(* Logix 5000 project; controller OptixProdData_Demo vendor 1 type 14 code 164 rev 37.11; software revision 37.00 *)

TASK MainTask (continuous, watchdog 500 ms) : MainProgram

MODULES
   Local : vendor 1 type 14 code 164 (ICP 0, rev 37.11)
END_MODULES

TYPE str_01 :
STRUCT
   LEN : DINT;
   DATA : SINT[1];
END_STRUCT
END_TYPE

TYPE str_50 :   // String with 50 Characters for SQL Stored Procedures
STRUCT
   LEN : DINT;
   DATA : SINT[50];
END_STRUCT
END_TYPE

TYPE str_Date :
STRUCT
   LEN : DINT;
   DATA : SINT[12];
END_STRUCT
END_TYPE

TYPE str_DateTime :
STRUCT
   LEN : DINT;
   DATA : SINT[22];
END_STRUCT
END_TYPE

TYPE str_Time :
STRUCT
   LEN : DINT;
   DATA : SINT[10];
END_STRUCT
END_TYPE

TYPE udt_CycleTimes :
STRUCT
   ProdLine : str_50;   // Production Line Name
   StationID : str_50;   // Station Name
   TS_PLC : str_DateTime;   // PLC Time Stamp in DateTime format "01/01/2025 15:01:01"
   CycleTime : REAL;   // Cycle time in decimal seconds
   CycleTimeAvg : REAL;   // Cycle Time Average for last hour in deimal seconds
   CycleCount : DINT;   // non-reset Cycle Count
END_STRUCT
END_TYPE

TYPE udt_DateTime :   // WallClock structure
STRUCT
   Year : DINT;   // 2xxx
   Month : DINT;   // 1 - 12
   Day : DINT;   // 01 - 31
   Hour : DINT;   // 0 - 23
   Minute : DINT;   // 0 - 59
   Seconds : DINT;   // 0 - 59
   ms : DINT;   // 0 - 999,999
END_STRUCT
END_TYPE

TYPE udt_LineSummary :   // Summary production data to mimic existing white board
STRUCT
   ProdLine : str_50;   // Production Line Name
   Hour : str_Time;   // 24-hour clock time format HH:MM:SS
   Date : str_Date;   // Date in format 01/01/2025
   TargetQty : DINT;   // Target Qty for hour
   ActQty : DINT;   // Actual qty for hour
   TargetAccQty : DINT;   // Target Accumulated Qty
   ActAccQty : DINT;   // Actual Accumulated Qty
END_STRUCT
END_TYPE

TYPE udt_ProdData :   // Summary production data to mimic existing white board
STRUCT
   PLC_TS : str_DateTime;   // Controller Date Time "HH:MM:SS 01/25/2025"
   ProdLine : str_50;   // Production Line Name
   EquipID : str_50;   // Equipment Name
   ProdCount : DINT;   // Production Counter
   CycleAvg : REAL;   // Average Cycle time (seconds per part)
END_STRUCT
END_TYPE

TYPE udt_SPInterface :
STRUCT
   Trans_DN : BOOL;   // Transaction Complete Bit from Optix to PLC
   SQLErrorNum : DINT;   // SQL Error Number if transaction failed
   Trigger : DINT;   // DINT Value to increment to trigger stored procedure in Optix
END_STRUCT
END_TYPE

ADD_ON_INSTRUCTION ParseTime_SQL   (* revision 1.0 *)
VAR_IN_OUT
   TimeStamp : udt_DateTime; {required}
   Date : str_Date; {required}
   Time : str_Time; {required}
   DateTime : str_DateTime; {required}
END_VAR
VAR
   strTemp2 : str_DateTime; {access None}
   strTemp1 : str_DateTime; {access None}
   strTemp : str_DateTime; {access None}
   strYear : str_Date; {access None}
   strDateTime : str_DateTime; {access None}
   strDate : str_Date; {access None}
   strTime : str_Time; {access None}
END_VAR

ROUTINE Logic   (* structured text *)
   DTOS(TimeStamp.Year, strYear);
   //Create Time format
   #region
   //Hour
   IF TimeStamp.Hour<10 then
   	strTemp1:='0';
   	DTOS(TimeStamp.Hour, strTemp2);
   	CONCAT(strTemp1, strTemp2, strTemp);
   	//0h
   else
   	DTOS(TimeStamp.Hour,strTemp);
   	//hh
   end_if;
   
   strTemp1:=':';
   CONCAT(strTemp, strTemp1, strTime);
   //hh:
   
   //Minutes
   IF TimeStamp.Minute<10 then
   	strTemp1:='0';
   	DTOS(TimeStamp.Minute, strTemp2);
   	CONCAT(strTemp1, strTemp2, strTemp);
   	//0m
   else
   	DTOS(TimeStamp.Minute,strTemp);
   	//mm
   end_if;
   
   strTemp1:=':';
   CONCAT(strTime, strTemp, strTime);
   CONCAT(strTime, strTemp1, strTime);
   //hh:mm:
   //Seconds
   IF TimeStamp.Seconds<10 then
   	strTemp1:='0';
   	DTOS(TimeStamp.Seconds, strTemp2);
   	CONCAT(strTemp1, strTemp2, strTemp);
   	//0n
   else
   	DTOS(TimeStamp.Seconds,strTemp);
   	//nn
   end_if;
   #endregion
   //Time
   CONCAT(strTime, strTemp,strTime);
   //hh:mm:ss
   
   //Build Date
   #region
   //Month
   IF TimeStamp.Month<10 then
   	strTemp1:='0';
   	DTOS(TimeStamp.Month, strTemp2);
   	CONCAT(strTemp1, strTemp2, strTemp);
   	//0n
   else
   	DTOS(TimeStamp.Month,strTemp);
   	//mm
   end_if;
   
   strTemp1:='/';
   CONCAT(strTemp, strTemp1, strDate);
   //mm/
   
   //Day
   IF TimeStamp.Day<10 then
   	strTemp1:='0';
   	DTOS(TimeStamp.Day, strTemp2);
   	CONCAT(strTemp1, strTemp2, strTemp);
   	//0d
   else
   	DTOS(TimeStamp.Day,strTemp);
   	//dd
   end_if;
   strTemp1:='/';
   CONCAT(strDate, strTemp, strDate);
   CONCAT(strDate, strTemp1, strDate);
   //mm/dd/
   #endregion
   //Year
   CONCAT(strDate,strYear, strDate);
   //mm/dd/yyyy
   
   //Build DateTime
   
   strTemp := ' ';
   
   CONCAT(strDate, strTemp, strDateTime);
   CONCAT(strDateTime, strTime, strDateTime);
   
   //Need to use synchronous copy to prevent invallid data time structures
   CPS(strTime, Time, 1);
   CPS(strDate, Date, 1);
   CPS(strDateTime, DateTime, 1);
   
END_ROUTINE
END_ADD_ON_INSTRUCTION

VAR_GLOBAL   (* controller tags *)
   EmptyFile : BOOL;
   gONS : BOOL[320];   // Global One Shots
   Line1Buff_Ctl : CONTROL := (LEN := 200, EM := 1);
   Line1CycleAvg : REAL := 23.251;
   Line1Depalletizer1LD : BOOL;
   Line1Name : str_50 := 'Line - 1';
   Line1ProdCount : DINT := 325;
   Line1Station1 : str_50 := 'Depalletizer - 01';
   Line1Summary_Buffer : udt_ProdData[200];
   Line1Summary_LD : udt_ProdData := (PLC_TS := '06/17/2025 17:02:49', ProdLine := 'Line - 1', EquipID := 'Depalletizer - 01', ProdCount := 325, CycleAvg := 23.251);
   Line1SummaryDB_LD : udt_ProdData := (PLC_TS := '06/17/2025 17:01:54', ProdLine := 'Line - 1', EquipID := 'Depalletizer - 01', ProdCount := 325, CycleAvg := 23.251);
   SPLine1Summary : udt_SPInterface := (Trigger := 2366);
   strDateNow : str_Date := '06/17/2025';
   strDateTimeNow : str_DateTime := '06/17/2025 17:02:49';
   strTimeNow : str_Time := '17:02:49';
   strTimeStamps : ParseTime_SQL;
   TimeNow : udt_DateTime := (Year := 2025, Month := 6, Day := 17, Hour := 17, Minute := 2, Seconds := 49, ms := 705845);
   tmrFFUSummaryL1 : TIMER := (PRE := 1000);
   tmrTriggerSummaryL1 : TIMER := (PRE := 1000);
   UnloadLine1Summary : BOOL;
END_VAR

PROGRAM MainProgram   (* main routine MainRoutine *)

ROUTINE DateTime   (* ladder *)
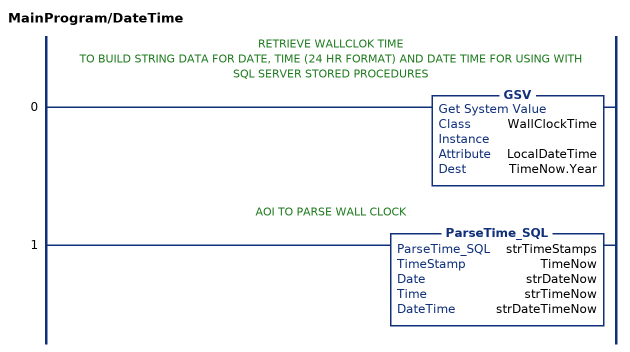
   // RETRIEVE WALLCLOK TIME
   // TO BUILD STRING DATA FOR DATE, TIME (24 HR FORMAT) AND DATE TIME FOR USING WITH SQL SERVER STORED PROCEDURES
   0: GSV(WallClockTime,,LocalDateTime,TimeNow.Year);
   // AOI TO PARSE WALL CLOCK
   1: ParseTime_SQL(strTimeStamps,TimeNow,strDateNow,strTimeNow,strDateTimeNow);
END_ROUTINE

ROUTINE LoadSummary   (* ladder *)
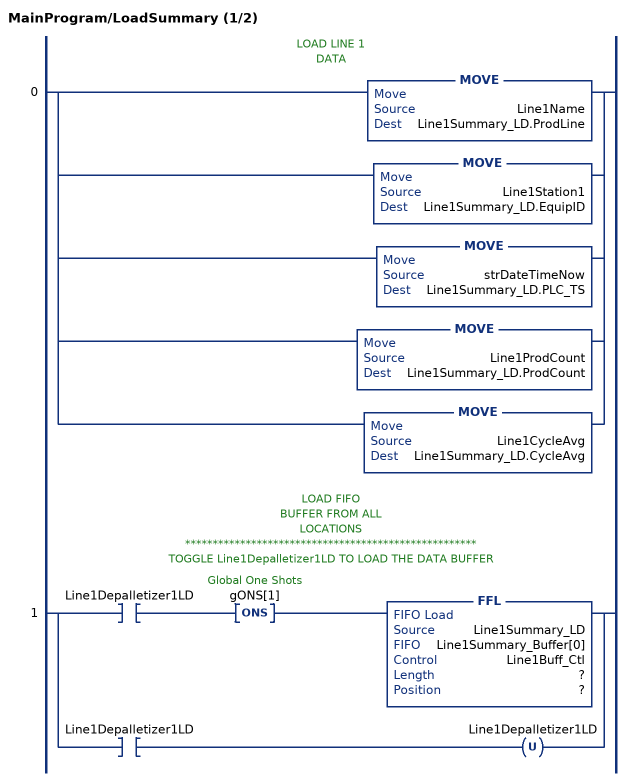
   // LOAD LINE 1
   // DATA
   0: [MOVE(Line1Name,Line1Summary_LD.ProdLine) ,MOVE(Line1Station1,Line1Summary_LD.EquipID) ,MOVE(strDateTimeNow,Line1Summary_LD.PLC_TS) ,MOVE(Line1ProdCount,Line1Summary_LD.ProdCount) ,MOVE(Line1CycleAvg,Line1Summary_LD.CycleAvg) ];
   // LOAD FIFO
   // BUFFER FROM ALL
   // LOCATIONS
   // *****************************************************
   // TOGGLE Line1Depalletizer1LD TO LOAD THE DATA BUFFER
   1: [XIC(Line1Depalletizer1LD) ONS(gONS[1]) FFL(Line1Summary_LD,Line1Summary_Buffer[0],Line1Buff_Ctl,?,?) ,XIC(Line1Depalletizer1LD) OTU(Line1Depalletizer1LD) ];
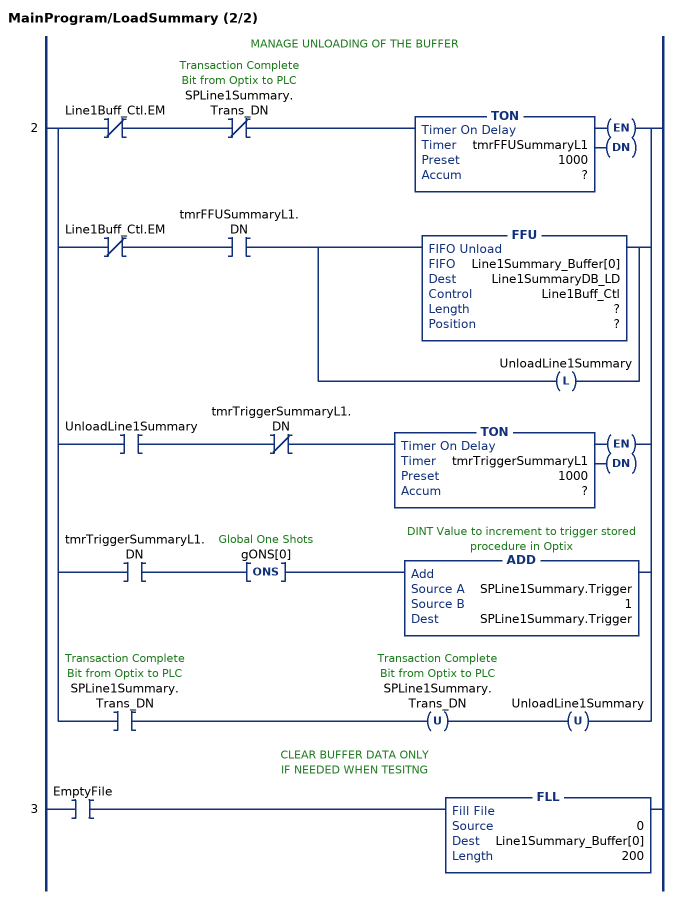
   // MANAGE UNLOADING OF THE BUFFER
   2: [XIO(Line1Buff_Ctl.EM) XIO(SPLine1Summary.Trans_DN) TON(tmrFFUSummaryL1,?,?) ,XIO(Line1Buff_Ctl.EM) XIC(tmrFFUSummaryL1.DN) [FFU(Line1Summary_Buffer[0],Line1SummaryDB_LD,Line1Buff_Ctl,?,?) ,OTL(UnloadLine1Summary) ] ,XIC(UnloadLine1Summary) XIO(tmrTriggerSummaryL1.DN) TON(tmrTriggerSummaryL1,?,?) ,XIC(tmrTriggerSummaryL1.DN) ONS(gONS[0]) ADD(SPLine1Summary.Trigger,1,SPLine1Summary.Trigger) ,XIC(SPLine1Summary.Trans_DN) OTU(SPLine1Summary.Trans_DN) OTU(UnloadLine1Summary) ];
   // CLEAR BUFFER DATA ONLY
   // IF NEEDED WHEN TESITNG
   3: XIC(EmptyFile)FLL(0,Line1Summary_Buffer[0],200);
END_ROUTINE

ROUTINE MainRoutine   (* ladder *)
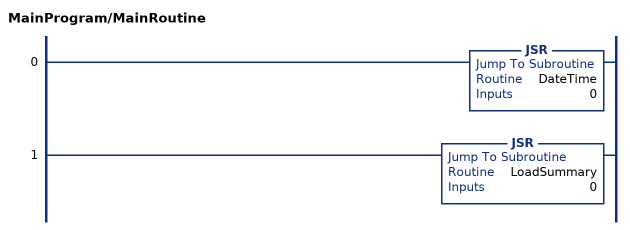
   0: JSR(DateTime,0);
   1: JSR(LoadSummary,0);
END_ROUTINE
END_PROGRAM
